(* IEC 61131-3 sources: AXOpen/src/template.axolibrary/ctrl/test, 2 files *)

(* ---- CylinderTests.st ---- *)
USING AXOpen.Core;
USING AXOpen.Rtc;
USING AXOpen.Logging;

NAMESPACE Template.Axolibrary.Tests
    {S7.extern=ReadWrite}
    CLASS TestContext IMPLEMENTS AXOpen.Core.IAxoContext
        VAR
            _openCounter : ULINT;
            _closeCounter : ULINT;
        END_VAR

        METHOD PUBLIC Open : ULINT
            _openCounter := _openCounter + ULINT#1;
        END_METHOD

        METHOD PUBLIC Close : ULINT
            _closeCounter := _closeCounter + ULINT#1;
        END_METHOD

        METHOD PUBLIC CreateIdentity : ULINT
            ;
        END_METHOD

        METHOD PUBLIC OpenCycleCount : ULINT
            OpenCycleCount := _openCounter;
        END_METHOD

        METHOD PUBLIC GetRtc : AXOpen.Rtc.IAxoRtc
            ;
        END_METHOD

        METHOD PUBLIC InjectRtc
            VAR_INPUT
                Rtc : IAxoRtc;
            END_VAR

            ;
        END_METHOD

        METHOD PUBLIC GetLogger : IAxoLogger
            ;
        END_METHOD

        METHOD PUBLIC InjectLogger
            VAR_INPUT
                _logger : IAxoLogger;
            END_VAR

            ;
        END_METHOD
    END_CLASS
    {TestFixture}
    {S7.extern=ReadWrite}
    CLASS CylinderTests
        VAR
            context : TestContext;
            cylinder : TemplateComponent;
            _homeSensor : BOOL;
            _workSensor : BOOL;
            _moveHomeSignal : BOOL;
            _moveWorkSignal : BOOL;
            _done : BOOL;
        END_VAR
        {Test}
        METHOD PUBLIC MoveHome
            WHILE _done DO
                context.Open();
                _done := Cylinder.MoveToHome().IsDone();
                cylinder.Run(context, WORD#64, REF(_homeSensor), REF(_workSensor), REF(_moveHomeSignal), REF(_moveWorkSignal));
                AxUnit.Assert.Equal(_moveHomeSignal, _moveHomeSignal);
                context.Close();
            END_WHILE;
        END_METHOD
    END_CLASS
END_NAMESPACE

(* ---- TemplateTests.st ---- *)
USING AXUnit;
USING AXOpen.Core;
USING AXOpen.Core.Dummies;
USING AXOpen.Rtc;
USING AXOpen.Rtm;
USING AXOpen.Logging;
USING Template.Axolibrary;

NAMESPACE Template.Axolibrary.Tests
    {S7.extern=ReadWrite}
    CLASS TestContext EXTENDS AXOpen.Core.Dummies.MockAxoContext
            METHOD PROTECTED OVERRIDE Main
                ;
            END_METHOD
    END_CLASS
    {TestFixture}
    {S7.extern=ReadWrite}
    CLASS CylinderTests
        VAR PROTECTED
            _context        :   TestContext;
            _rootObject     :   MockAxoObject;
            _component      :   Template.Axolibrary.TemplateComponent;
        END_VAR

        VAR PRIVATE
            _contextClean    :   TestContext;
            _rtc             :   AXOpen.Core.Dummies.MockAxoRtc;
            _rtm             :   AXOpen.Core.Dummies.MockAxoRtm;
        END_VAR

        {TestSetup}
        METHOD PUBLIC TestSetup
            _context    :=  _contextClean;
            _context.InitializeRootObject(_rootObject);
            _rtm.SetElapsed(LTIME#2s);
            _context.InjectRtm(_rtm);
            _rtc.SetNowUTC(LDATE_AND_TIME#2012-01-12-15:58:12.123);
            _context.InjectRtc(_rtc);
        END_METHOD

        {Test}
        METHOD PUBLIC MoveHome
            _context.Open();
            THIS._component.Run(
                                parent  :=   _rootObject,
                                hwID    :=   UINT#60);
            AxUnit.Assert.Equal(TRUE, TRUE);
            _context.Close();
    END_METHOD
    END_CLASS
END_NAMESPACE
